FUNCTION HLI3_GetIpoState : BOOL
VAR_INPUT
	nChanIdx: INT;
END_VAR



IF NOT HLI3_CheckChannelValid(nChannel := nChanIdx) THEN
	RETURN;
END_IF

HLI3_GetIpoState:=gpCh[nChanIdx]^.bahn_state.interpolation_active_r;

END_FUNCTION

(* stored: Version 1.1.0.1, ProductVersion 3.1.0.12
   POU HLI3_GetIpoState: Id {71e85e22-595d-4b23-91f7-c7b0954e79a6} *)
